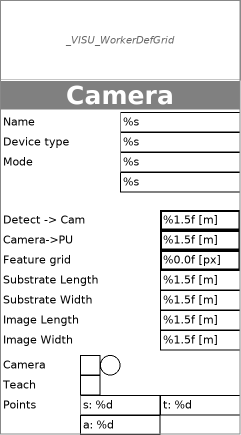
VISUALIZATION _VISU_WorkerDefGrid_Camera  // 241x435
VAR_IN_OUT
		m_Inst : FB_WorkerDefGrid_Camera;
END_VAR
    Frame (0,0 241x80)
        shows _VISU_WorkerDefGrid(m_Inst := m_Inst)
    Rectangle (80,395 80x20), "s: %d", tooltip "scanned points", text variable: m_Inst._nScannedPoints, invisible if: NOT m_Inst._bCamValid
    Rectangle (0,395 80x20), "Points"
    Rectangle (160,395 80x20), "t: %d", tooltip "teached points", text variable: m_Inst._nTeachedPoints, invisible if: NOT m_Inst._bCamValid
    Rectangle (0,355 80x20), "Camera"
    RoundedRectangle (80,355 20x20), colour toggle: m_Inst._bCamReady, invisible if: NOT m_Inst._bCamValid
    Rectangle (0,375 80x20), "Teach"
    RoundedRectangle (80,375 20x20), colour toggle: m_Inst._bTeachOk, invisible if: NOT m_Inst._bCamValid
    Rectangle (0,210 160x20), "Detect -> Cam"
    Rectangle (160,210 80x20), "%1.5f [m]", text variable: m_Inst._iActiveCam.fDetectToCameraOffset, invisible if: NOT m_Inst._bCamValid
        OnMouseClick: write the text variable via Default
    Rectangle (0,270 160x20), "Substrate Length"
    Rectangle (160,270 80x20), "%1.5f [m]", text variable: m_Inst._iActiveCam.fSubstrateLength, invisible if: NOT m_Inst._bCamValid
    Rectangle (0,230 160x20), "Camera->PU"
    Rectangle (160,230 80x20), "%1.5f [m]", text variable: m_Inst._iActiveCam.fCameraToPrintOffset, invisible if: NOT m_Inst._bCamValid
        OnMouseClick: write the text variable via Default
    Rectangle (0,80 240x30), "Camera", colour toggle: m_Inst._pAttachedCt <> 0
        OnMouseClick: change screen: AssignExpression m_Inst._iActiveCam.sVisuName
    Rectangle (80,415 80x20), "a: %d", tooltip "added points", text variable: m_Inst._nAddedPoint, invisible if: NOT m_Inst._bCamValid
    Rectangle (0,250 160x20), "Feature grid"
    Rectangle (160,250 80x20), "%0.0f [px]", text variable: m_Inst._fFeatureGrid, invisible if: NOT m_Inst._bCamValid
        OnMouseDown: write the text variable via Default
    Ellipse (100,355 20x20), tooltip "cam simulation", invisible if: NOT m_Inst._bCamValid
        toggle m_Inst._iActiveCam.bSimulate
    Rectangle (120,112 120x20), "%s", tooltip "active camera device", text variable: m_Inst._iActiveCam.sName
    Rectangle (120,172 120x20), "%s", tooltip "current camera mode (active cam)", text variable: m_Inst._iActiveCam.eCameraMode, colour toggle: m_Inst._pAdsCam^.stAds.eI_CameraMode <> m_Inst._iActiveCam.eCameraMode
    Rectangle (0,290 160x20), "Substrate Width"
    Rectangle (160,290 80x20), "%1.5f [m]", text variable: m_Inst._iActiveCam.fSubstrateWidth, invisible if: NOT m_Inst._bCamValid
    Rectangle (0,310 160x20), "Image Length"
    Rectangle (160,310 80x20), "%1.5f [m]", text variable: m_Inst._iActiveCam.fImageLength, invisible if: NOT m_Inst._bCamValid
    Rectangle (0,330 160x20), "Image Width"
    Rectangle (160,330 80x20), "%1.5f [m]", text variable: m_Inst._iActiveCam.fImageWidth, invisible if: NOT m_Inst._bCamValid
    Rectangle (120,152 120x20), "%s", tooltip "camera mode desired (active cam)", text variable: m_Inst._pAdsCam^.stAds.eI_CameraMode
    Rectangle (120,132 120x20), "%s", tooltip "active camera device type", text variable: m_Inst._iActiveCam.eDeviceType
    Rectangle (0,112 120x20), "Name"
    Rectangle (0,132 120x20), "Device type"
    Rectangle (0,152 120x20), "Mode"
END_VISUALIZATION

(* stored: Version 1.1.0.1, ProductVersion 3.1.4024.11
   Visu _VISU_WorkerDefGrid_Camera: Id {6da48dd2-d468-46e7-9518-8f2152f9bdb4} *)
